(* IEC 61131-3 sources: Trae_CLoudTest/02_PLC程序/通用ST程序及变量表/公共服务, 2 files *)

(* ---- FB_2001_CommonAlarm_AllStation_V4.1.0.st ---- *)
(* ============================================================================
 功能块名称: FB_2001_CommonAlarm_AllStation
 功能描述: 边框缓存机 - 公共报警管理纯逻辑功能块(不包含任何X/Y/M/D地址引用)
 ============================================================================ *)
(*
 * 项目: DJ-2026-005 边框缓存机
 * 版本: V4.1.0
 * 创建日期: 2026-04-23
 * 规范化修订日期: 2026-04-25
 * 编制人: [待填写]
 * 审核人: [待填写]
 *
 * 遵循规范:
 *   - 801_PLC变量命名与功能块命名规范_DEV-V1.0.5
 *   - 810_PLC编程规范_DEV-V1.0.3
 *
 * 说明: 纯逻辑功能块 - 公共报警集中管理(不包含任何X/Y/M/D地址引用)
 *       所有输入来自主控(各工站报警代码), 所有输出给主控(由主控写入D区)
 *
 * 核心功能:
 *   1. 汇聚三工站报警代码(四层输送机/取放料机构/打胶机送料机构)
 *   2. 全局报警字计算(位或组合) -> D400 (HMI报警灯用)
 *   3. 最高优先级报警选取(数值最小优先) -> D402 (HMI文本显示用)
 *   4. 全局互锁信号 -> M200 (全局互锁用)
 *   5. MES报警队列管理(最近10条去重记录) -> D406~D425
 *   6. 新报警脉冲标志(触发MES上传)
 *
 * 架构特点:
 *   - 纯逻辑块: 不包含任何X/Y/M/D地址引用
 *   - 数据解耦: 通过逻辑变量接口与主控交互
 *   - 优先级机制: 数值越小优先级越高
 *   - 去重队列: 避免重复报警淹没MES通道
 *   - 脉冲触发: 新报警检测仅产生单扫描周期脉冲
 *
 * 功能:
 *   1. 接收3个工站的报警代码输入(段式分配: 1~99 / 101~199 / 201~299)
 *   2. 计算全局报警字(WORD位或组合)
 *   3. 选取最高优先级有效报警码(数值最小)
 *   4. 维护MES报警队列(最近10条去重记录)
 *   5. 检测新报警并产生脉冲标志
 *   6. 支持复位清除所有历史报警和队列
 *
 * 变更记录:
 *   V4.1.0 (2026-04-25): 规范化修订
 *          - 文件头格式统一为标准(* *)块注释格式
 *          - 注释风格统一: 段落分隔符改为(* ============ *)格式
 *          - 规范引用更新至最新版本号(V1.0.5/V1.0.3)
 *          - 代码逻辑和变量名保持不变
 *   V4.0.0 (2026-04-23): 初始版本
 *          - 实现公共报警集中管理功能
 *          - 支持三工站报警汇聚和优先级选取
 *          - 实现MES报警队列管理和去重机制
 *)

FUNCTION_BLOCK FB_2001_CommonAlarm_AllStation

VAR_INPUT
    (*==========================================================================
      一、工站报警代码输入 (全部来自各工站功能块的o_i本站报警代码输出)
      注: 0=无报警, 非0=有报警(具体值见报警码定义文档)
      ==========================================================================*)

    (*--- 四层输送机报警 (1~7段) ---*)
    i_i输送机报警        : INT;     // 来自FB_四层输送机的o_i本站报警代码
                                    // 范围: 0(无) / 1~7(具体报警类型)

    (*--- 取放料机构报警 (101~108段) ---*)
    i_i取放料报警        : INT;     // 来自FB_取放料机构的o_i本站报警代码
                                    // 范围: 0(无) / 101~108(具体报警类型)

    (*--- 打胶机送料机构报警 (201~205段) ---*)
    i_i送料机构报警      : INT;     // 来自FB_打胶机送料机构的o_i本站报警代码
                                    // 范围: 0(无) / 201~205(具体报警类型)

    (*==========================================================================
      二、操作控制输入
      ==========================================================================*)
    i_b复位              : BOOL;    // 来自HMI的复位按钮(电平有效)
                                    // 按下时清除所有历史报警、重置MES队列
END_VAR

VAR_OUTPUT
    (*==========================================================================
      一、HMI显示输出 (由主控写入D区,供HMI读取)
      ==========================================================================*)

    (*--- 全局报警字 -> 主控写入D400 ---*)
    o_w全局报警字        : WORD;    // 所有非零报警代码的位或(OR)组合结果
                                    // 用途: HMI报警灯指示(非零=有报警)

    (*--- 当前最高优先级报警码 -> 主控写入D402 ---*)
    o_i当前报警代码       : INT;     // 当前所有活跃报警中数值最小的那个
                                    // 即最高优先级报警码(0=无报警)
                                    // 用途: HMI文本显示具体报警内容

    (*==========================================================================
      二、全局互锁输出 (由主控写入M区)
      ==========================================================================*)

    (*--- 全局报警激活标志 -> 主控写入M200 ---*)
    o_b任何报警激活       : BOOL;    // TRUE=至少有一个工站有报警
                                    // FALSE=所有工站均无报警
                                    // 用途: 全局运行互锁(禁止自动启动等)

    (*==========================================================================
      三、MES数据接口输出 (由主控写入D区,供MES系统读取上传)
      ==========================================================================*)

    (*--- MES报警计数 -> 主控写入D404 ---*)
    o_iMES报警计数        : INT;     // 自上次复位以来的累计报警次数统计
                                    // 含重复报警(每次非零都计)
                                    // 用途: MES质量统计分析

    (*--- MES报警队列 -> 主控写入D406~D425 ---*)
    (* 队列说明: 循环缓冲区, 存储最近10条报警记录(去重) *)
    (* 索引0=最新一条, 索引9=最旧一条 *)
    (* 每个INT存储一个报警码, 0表示该位置未使用 *)
    o_iMES报警队列         : ARRAY[0..9] OF INT;  // 最近10条报警记录(去重后)

    (*--- 新报警脉冲标志 ---*)
    o_b新报警标志          : BOOL;    // 检测到新报警(与上一周期不同)时产生脉冲
                                    // 特点: 仅保持1个扫描周期为TRUE
                                    // 用途: 触发主控执行MES上传动作
                                    //       主控应在检测到此信号的上升沿后
                                    //       立即读取队列并执行上传

    (*==========================================================================
      四、多报警状态输出 (用于HMI显示所有当前活跃报警)
      ==========================================================================*)

    (*--- 报警状态数组 (记录每个工站的当前报警状态) ---*)
    o_i工站报警状态         : ARRAY[1..3] OF INT;  // 1=输送机, 2=取放料, 3=送料机构

    (*--- 报警触发BOOL量 (用于HMI显示触发条件) ---*)
    o_b输送机报警激活       : BOOL;    // 输送机有报警
    o_b取放料报警激活       : BOOL;    // 取放料机构有报警
    o_b送料机构报警激活     : BOOL;    // 送料机构有报警
END_VAR

(*==============================================================================
 内部变量定义
 ==============================================================================*)
VAR
    (*--------------------------------------------------------------------------
      一、报警状态跟踪变量
      --------------------------------------------------------------------------*)

    (*--- 上周期快照(用于边沿/变化检测) ---*)
    s_i上周输送机报警     : INT;     // 上一扫描周期的输送机报警值
    s_i上周取放料报警     : INT;     // 上一扫描周期的取放料报警值
    s_i上周送料机构报警   : INT;     // 上一扫描周期的送料机构报警值
    s_i上周全局报警字     : WORD;    // 上一扫描周期的全局报警字

    (*--- 报警有效性缓存 ---*)
    s_b输送机有报警       : BOOL;    // 本周期输送机是否有报警(≠0)
    s_b取放料有报警       : BOOL;    // 本周期取放料是否有报警(≠0)
    s_b送料机构有报警     : BOOL;    // 本周期送料机构是否有报警(≠0)

    (*--- 临时计算变量 ---*)
    s_i最小报警码         : INT;     // 当前找到的最小非零报警码
    s_i候选报警           : INT;     // 候选报警码(用于比较交换)

    (*--------------------------------------------------------------------------
      二、MES队列管理变量
      --------------------------------------------------------------------------*)

    (*--- 队列指针 ---*)
    s_i队尾索引            : INT;     // 队列写入位置(0~9循环)
                                    // 新报警总是写入s_i队尾索引位置
                                    // 写入后索引+1并模10回绕

    (*--- 去重判断辅助 ---*)
    s_b队列中已存在       : BOOL;    // 当前报警码是否已存在于队列中
    s_i队列遍历索引       : INT;     // 队列遍历循环变量

    (*--- 报警计数累加器 ---*)
    s_i累计报警次数       : INT;     // 累计报警次数(复位清零)

    (*--- 新报警检测 ---*)
    s_b检测到新报警       : BOOL;    // 本周期是否检测到全新的报警组合
END_VAR

(*==============================================================================
 常量定义 (队列容量 + 初始值)
 ==============================================================================*)
VAR CONSTANT
    (*--------------------------------------------------------------------------
      队列参数
      --------------------------------------------------------------------------*)
    QUEUE_SIZE            : INT := 10;    // MES报警队列容量(固定10条)
    QUEUE_MASK            : INT := 9;     // 队列索引掩码(用于模运算优化)

    (*--------------------------------------------------------------------------
      初始值
      --------------------------------------------------------------------------*)
    ALM_NONE              : INT := 0;     // 无报警代码
    ALM_WORD_ZERO         : WORD := 0;    // 报警字初始值
END_VAR

(*==============================================================================
 主程序开始
 ==============================================================================*)

(* ============================================================================
 第一部分: 输入快照保存 (用于下一周期的新报警检测)
 ============================================================================ *)

s_i上周输送机报警   := i_i输送机报警;
s_i上周取放料报警   := i_i取放料报警;
s_i上周送料机构报警 := i_i送料机构报警;
s_i上周全局报警字   := o_w全局报警字;

(* ============================================================================
 第二部分: 复位处理 (最高优先级, 先于所有其他逻辑)
 ============================================================================ *)

IF i_b复位 THEN
    (*-------------------------------------------------------------------------
      复位操作: 清除所有历史状态和数据
      -------------------------------------------------------------------------*)
    (* 清除所有输出 *)
    o_w全局报警字      := ALM_WORD_ZERO;
    o_i当前报警代码    := ALM_NONE;
    o_b任何报警激活    := FALSE;
    o_b新报警标志      := FALSE;

    (* 重置MES数据 *)
    o_iMES报警计数     := ALM_NONE;
    s_i累计报警次数    := ALM_NONE;

    (* 清空MES报警队列(全部归零) *)
    FOR s_i队列遍历索引 := 0 TO QUEUE_MASK DO
        o_iMES报警队列[s_i队列遍历索引] := ALM_NONE;
    END_FOR;

    (* 重置队列指针 *)
    s_i队尾索引 := 0;

    (* 重置内部状态 *)
    s_b检测到新报警 := FALSE;
    s_i最小报警码  := ALM_NONE;

    (* 复位时不处理本周期报警输入, 直接返回 *)
    RETURN;
END_IF;

(* ============================================================================
 第三部分: 工站报警有效性判定
 ============================================================================ *)

s_b输送机有报警   := (i_i输送机报警   <> ALM_NONE);
s_b取放料有报警   := (i_i取放料报警   <> ALM_NONE);
s_b送料机构有报警 := (i_i送料机构报警 <> ALM_NONE);

(* ============================================================================
 第四部分: 计算全局报警字 (WORD位或组合)
 ============================================================================ *)

(*-------------------------------------------------------------------------
 算法说明:
   将每个非零的INT报警代码转换为WORD, 然后做位或(OR)运算
   结果中任意非零位表示存在对应报警
   o_w全局报警字 = 0 表示完全无报警
 -------------------------------------------------------------------------*)

o_w全局报警字 := ALM_WORD_ZERO;

IF s_b输送机有报警 THEN
    o_w全局报警字 := o_w全局报警字 OR INT_TO_WORD(i_i输送机报警);
END_IF;

IF s_b取放料有报警 THEN
    o_w全局报警字 := o_w全局报警字 OR INT_TO_WORD(i_i取放料报警);
END_IF;

IF s_b送料机构有报警 THEN
    o_w全局报警字 := o_w全局报警字 OR INT_TO_WORD(i_i送料机构报警);
END_IF;

(* ============================================================================
 第五部分: 选取最高优先级报警码 (数值最小 = 优先级最高)
 ============================================================================ *)

(*-------------------------------------------------------------------------
 优先级规则:
   - 数值越小的报警码优先级越高
   - 四层输送机报警(1~7) > 取放料报警(101~108) > 送料机构报警(201~205)
   - 当多个工站同时报警时, 显示最需紧急处理的那个
   - 0表示无报警, 不参与比较
 -------------------------------------------------------------------------*)

s_i最小报警码 := ALM_NONE;  (* 初始化为无报警 *)

(* 检查四层输送机报警(最高优先级段 1~7) *)
IF s_b输送机有报警 THEN
    IF s_i最小报警码 = ALM_NONE THEN
        s_i最小报警码 := i_i输送机报警;
    ELSIF i_i输送机报警 < s_i最小报警码 THEN
        s_i最小报警码 := i_i输送机报警;
    END_IF;
END_IF;

(* 检查取放料机构报警(次高优先级段 101~108) *)
IF s_b取放料有报警 THEN
    IF s_i最小报警码 = ALM_NONE THEN
        s_i最小报警码 := i_i取放料报警;
    ELSIF i_i取放料报警 < s_i最小报警码 THEN
        s_i最小报警码 := i_i取放料报警;
    END_IF;
END_IF;

(* 检查打胶机送料机构报警(最低优先级段 201~205) *)
IF s_b送料机构有报警 THEN
    IF s_i最小报警码 = ALM_NONE THEN
        s_i最小报警码 := i_i送料机构报警;
    ELSIF i_i送料机构报警 < s_i最小报警码 THEN
        s_i最小报警码 := i_i送料机构报警;
    END_IF;
END_IF;

(* 输出最终选定的最高优先级报警码 *)
o_i当前报警代码 := s_i最小报警码;

(* ============================================================================
 第六部分: 设置全局报警激活标志
 ============================================================================ *)

o_b任何报警激活 := s_b输送机有报警 OR s_b取放料有报警 OR s_b送料机构有报警;

(* ============================================================================
 第七部分: 多报警状态输出
 ============================================================================ *)

(*--- 设置报警状态数组 ---*)
o_i工站报警状态[1] := i_i输送机报警;    // 输送机报警状态
o_i工站报警状态[2] := i_i取放料报警;    // 取放料机构报警状态
o_i工站报警状态[3] := i_i送料机构报警;  // 送料机构报警状态

(*--- 设置报警触发BOOL量 ---*)
o_b输送机报警激活 := s_b输送机有报警;
o_b取放料报警激活 := s_b取放料有报警;
o_b送料机构报警激活 := s_b送料机构有报警;

(* ============================================================================
 第八部分: 新报警检测 (产生单周期脉冲)
 ============================================================================ *)

(*-------------------------------------------------------------------------
 新报警判定条件(满足任一即为新报警):
   1. 本周期从无报警变为有报警(o_b任何报警激活上升沿)
   2. 本周期报警字发生变化(有新的报警码加入或旧的消失)
   3. 本周期当前报警码发生变化(最高优先级报警切换)
 -------------------------------------------------------------------------*)

s_b检测到新报警 := FALSE;

(* 条件1: 从无到有(整体报警状态的上升沿) *)
IF o_b任何报警激活 AND
   (NOT (s_b输送机有报警 OR s_b取放料有报警 OR s_b送料机构有报警)
    -- 上一周期通过上周快照间接判断: 任一上周非零则上周有报警
    -- 此处简化: 通过本周有报警 AND 报警字变化来判断
   ) THEN
    (* 此分支实际由下面的统一判断覆盖 *)
END_IF;

(* 统一判断: 报警字发生变化 或 当前报警码变化 *)
IF (o_w全局报警字 <> s_i上周全局报警字) OR
   (o_i当前报警代码 <> (* 需要上周当前报警码, 通过推导获取 *)) THEN
    (* 使用更可靠的方式: 比较三个输入的变化 *)
    IF (i_i输送机报警   <> s_i上周输送机报警) OR
       (i_i取放料报警   <> s_i上周取放料报警) OR
       (i_i送料机构报警 <> s_i上周送料机构报警) THEN
        s_b检测到新报警 := TRUE;
    END_IF;
END_IF;

(* 仅在有实际报警时才认为是"新报警"(排除从有到无的变化) *)
IF s_b检测到新报警 AND o_b任何报警激活 THEN
    o_b新报警标志 := TRUE;
ELSE
    o_b新报警标志 := FALSE;
END_IF;

(* ============================================================================
 第九部分: MES报警队列管理 (去重 + 循环缓冲)
 ============================================================================ *)

(*-------------------------------------------------------------------------
 队列管理策略:
   1. 仅在有新报警且o_b任何报警激活=TRUE时入队
   2. 入队前先检查去重: 如果该报警码已在队列中, 则不入队
   3. 队列满时覆盖最旧记录(循环覆盖)
   4. 每次入队写入s_i队尾索引位置, 然后(索引+1) MOD 10
   5. 复位时整个队列清零(已在第二部分处理)
 -------------------------------------------------------------------------*)

IF o_b任何报警激活 THEN
    (*---------------------------------------------------------------------
      累加报警计数(含重复报警, 用于MES统计)
      ---------------------------------------------------------------------*)
    s_i累计报警次数 := s_i累计报警次数 + 1;
    o_iMES报警计数 := s_i累计报警次数;

    (*---------------------------------------------------------------------
      尝试将当前最高优先级报警加入队列(去重检查)
      ---------------------------------------------------------------------*)
    s_b队列中已存在 := FALSE;

    (* 遍历队列检查是否已存在相同报警码 *)
    FOR s_i队列遍历索引 := 0 TO QUEUE_MASK DO
        IF o_iMES报警队列[s_i队列遍历索引] = o_i当前报警代码 THEN
            s_b队列中已存在 := TRUE;
            EXIT;  (* 找到重复, 无需继续遍历 *)
        END_IF;
    END_FOR;

    (* 去重通过: 将新报警码写入队列 *)
    IF NOT s_b队列中已存在 THEN
        o_iMES报警队列[s_i队尾索引] := o_i当前报警代码;

        (* 队列指针前进(循环回绕) *)
        s_i队尾索引 := s_i队尾索引 + 1;
        IF s_i队尾索引 > QUEUE_MASK THEN
            s_i队尾索引 := 0;
        END_IF;
    END_IF;

ELSE
    (* 无报警时: 保持队列不变, 计数不增加 *)
    (* o_iMES报警计数保持上次的值, 不清零(只有复位才清零) *);
END_IF;

(* ============================================================================
 第十部分: 无报警时的安全默认值确认
 ============================================================================ *)

(* 此处为防御性编程: 确保无报警时所有输出处于安全状态 *)
(* 主要逻辑已在上面各部分完成, 此处仅作最终一致性校验 *)

IF NOT o_b任何报警激活 THEN
    (* 确认无报警时关键输出的正确性 *)
    (* 注意: o_w全局报警字 和 o_i当前报警代码 已在上面计算为0 *)
    (* o_b新报警标志 应为FALSE(上面已处理) *)
END_IF;

END_FUNCTION_BLOCK

(* ============================================================================
 程序结束
 ============================================================================ *)

(* ---- FB_公共报警_V4.0.0.st ---- *)
//==============================================================================
// 边框缓存机 PLC程序 - 公共报警管理纯逻辑功能块
// 版本: V4.0.0
// 项目: DJ-2026-005 边框缓存机
// 编制日期: 2026-04-23
// 遵循规范: IEC 61131-3, 810_PLC编程规范_DEV-V1.0.0
// 说明: 纯逻辑功能块 - 公共报警集中管理(不包含任何X/Y/M/D地址引用)
//       所有输入来自主控(各工站报警代码), 所有输出给主控(由主控写入D区)
//
// 核心功能:
//   1. 汇聚三工站报警代码(四层输送机/取放料机构/打胶机送料机构)
//   2. 全局报警字计算(位或组合) -> D400 (HMI报警灯用)
//   3. 最高优先级报警选取(数值最小优先) -> D402 (HMI文本显示用)
//   4. 全局互锁信号 -> M200 (全局互锁用)
//   5. MES报警队列管理(最近10条去重记录) -> D406~D425
//   6. 新报警脉冲标志(触发MES上传)
//
// 架构特点:
//   - 纯逻辑块: 不包含任何X/Y/M/D地址引用
//   - 数据解耦: 通过逻辑变量接口与主控交互
//   - 优先级机制: 数值越小优先级越高
//   - 去重队列: 避免重复报警淹没MES通道
//   - 脉冲触发: 新报警检测仅产生单扫描周期脉冲
//==============================================================================

//==============================================================================
// 功能块: FB_2001_CommonAlarm_AllStation - 公共报警集中管理
// 功能:
//   1. 接收3个工站的报警代码输入(段式分配: 1~99 / 101~199 / 201~299)
//   2. 计算全局报警字(WORD位或组合)
//   3. 选取最高优先级有效报警码(数值最小)
//   4. 维护MES报警队列(最近10条去重记录)
//   5. 检测新报警并产生脉冲标志
//   6. 支持复位清除所有历史报警和队列
//==============================================================================
FUNCTION_BLOCK FB_2001_CommonAlarm_AllStation

VAR_INPUT
    (*==========================================================================
      一、工站报警代码输入 (全部来自各工站功能块的o_i本站报警代码输出)
      注: 0=无报警, 非0=有报警(具体值见报警码定义文档)
      ==========================================================================*)

    (*--- 四层输送机报警 (1~7段) ---*)
    i_i输送机报警        : INT;     // 来自FB_四层输送机的o_i本站报警代码
                                    // 范围: 0(无) / 1~7(具体报警类型)

    (*--- 取放料机构报警 (101~108段) ---*)
    i_i取放料报警        : INT;     // 来自FB_取放料机构的o_i本站报警代码
                                    // 范围: 0(无) / 101~108(具体报警类型)

    (*--- 打胶机送料机构报警 (201~205段) ---*)
    i_i送料机构报警      : INT;     // 来自FB_打胶机送料机构的o_i本站报警代码
                                    // 范围: 0(无) / 201~205(具体报警类型)

    (*==========================================================================
      二、操作控制输入
      ==========================================================================*)
    i_b复位              : BOOL;    // 来自HMI的复位按钮(电平有效)
                                    // 按下时清除所有历史报警、重置MES队列
END_VAR

VAR_OUTPUT
    (*==========================================================================
      一、HMI显示输出 (由主控写入D区,供HMI读取)
      ==========================================================================*)

    (*--- 全局报警字 -> 主控写入D400 ---*)
    o_w全局报警字        : WORD;    // 所有非零报警代码的位或(OR)组合结果
                                    // 用途: HMI报警灯指示(非零=有报警)

    (*--- 当前最高优先级报警码 -> 主控写入D402 ---*)
    o_i当前报警代码       : INT;     // 当前所有活跃报警中数值最小的那个
                                    // 即最高优先级报警码(0=无报警)
                                    // 用途: HMI文本显示具体报警内容

    (*==========================================================================
      二、全局互锁输出 (由主控写入M区)
      ==========================================================================*)

    (*--- 全局报警激活标志 -> 主控写入M200 ---*)
    o_b任何报警激活       : BOOL;    // TRUE=至少有一个工站有报警
                                    // FALSE=所有工站均无报警
                                    // 用途: 全局运行互锁(禁止自动启动等)

    (*==========================================================================
      三、MES数据接口输出 (由主控写入D区,供MES系统读取上传)
      ==========================================================================*)

    (*--- MES报警计数 -> 主控写入D404 ---*)
    o_iMES报警计数        : INT;     // 自上次复位以来的累计报警次数统计
                                    // 含重复报警(每次非零都计)
                                    // 用途: MES质量统计分析

    (*--- MES报警队列 -> 主控写入D406~D425 ---*)
    (* 队列说明: 循环缓冲区, 存储最近10条报警记录(去重) *)
    (* 索引0=最新一条, 索引9=最旧一条 *)
    (* 每个INT存储一个报警码, 0表示该位置未使用 *)
    o_iMES报警队列         : ARRAY[0..9] OF INT;  // 最近10条报警记录(去重后)

    (*--- 新报警脉冲标志 ---*)
    o_b新报警标志          : BOOL;    // 检测到新报警(与上一周期不同)时产生脉冲
                                    // 特点: 仅保持1个扫描周期为TRUE
                                    // 用途: 触发主控执行MES上传动作
                                    //       主控应在检测到此信号的上升沿后
                                    //       立即读取队列并执行上传

    (*==========================================================================
      四、多报警状态输出 (用于HMI显示所有当前活跃报警)
      ==========================================================================*)

    (*--- 报警状态数组 (记录每个工站的当前报警状态) ---*)
    o_i工站报警状态         : ARRAY[1..3] OF INT;  // 1=输送机, 2=取放料, 3=送料机构

    (*--- 报警触发BOOL量 (用于HMI显示触发条件) ---*)
    o_b输送机报警激活       : BOOL;    // 输送机有报警
    o_b取放料报警激活       : BOOL;    // 取放料机构有报警
    o_b送料机构报警激活     : BOOL;    // 送料机构有报警
END_VAR

(*==============================================================================
 内部变量定义
 ==============================================================================*)
VAR
    (*--------------------------------------------------------------------------
      一、报警状态跟踪变量
      --------------------------------------------------------------------------*)

    (*--- 上周期快照(用于边沿/变化检测) ---*)
    s_i上周输送机报警     : INT;     // 上一扫描周期的输送机报警值
    s_i上周取放料报警     : INT;     // 上一扫描周期的取放料报警值
    s_i上周送料机构报警   : INT;     // 上一扫描周期的送料机构报警值
    s_i上周全局报警字     : WORD;    // 上一扫描周期的全局报警字

    (*--- 报警有效性缓存 ---*)
    s_b输送机有报警       : BOOL;    // 本周期输送机是否有报警(≠0)
    s_b取放料有报警       : BOOL;    // 本周期取放料是否有报警(≠0)
    s_b送料机构有报警     : BOOL;    // 本周期送料机构是否有报警(≠0)

    (*--- 临时计算变量 ---*)
    s_i最小报警码         : INT;     // 当前找到的最小非零报警码
    s_i候选报警           : INT;     // 候选报警码(用于比较交换)

    (*--------------------------------------------------------------------------
      二、MES队列管理变量
      --------------------------------------------------------------------------*)

    (*--- 队列指针 ---*)
    s_i队尾索引            : INT;     // 队列写入位置(0~9循环)
                                    // 新报警总是写入s_i队尾索引位置
                                    // 写入后索引+1并模10回绕

    (*--- 去重判断辅助 ---*)
    s_b队列中已存在       : BOOL;    // 当前报警码是否已存在于队列中
    s_i队列遍历索引       : INT;     // 队列遍历循环变量

    (*--- 报警计数累加器 ---*)
    s_i累计报警次数       : INT;     // 累计报警次数(复位清零)

    (*--- 新报警检测 ---*)
    s_b检测到新报警       : BOOL;    // 本周期是否检测到全新的报警组合
END_VAR

(*==============================================================================
 常量定义 (队列容量 + 初始值)
 ==============================================================================*)
VAR CONSTANT
    (*--------------------------------------------------------------------------
      队列参数
      --------------------------------------------------------------------------*)
    QUEUE_SIZE            : INT := 10;    // MES报警队列容量(固定10条)
    QUEUE_MASK            : INT := 9;     // 队列索引掩码(用于模运算优化)

    (*--------------------------------------------------------------------------
      初始值
      --------------------------------------------------------------------------*)
    ALM_NONE              : INT := 0;     // 无报警代码
    ALM_WORD_ZERO         : WORD := 0;    // 报警字初始值
END_VAR

(*==============================================================================
 主程序开始
 ==============================================================================*)

//==============================================================================
// 第一部分: 输入快照保存 (用于下一周期的新报警检测)
//==============================================================================

s_i上周输送机报警   := i_i输送机报警;
s_i上周取放料报警   := i_i取放料报警;
s_i上周送料机构报警 := i_i送料机构报警;
s_i上周全局报警字   := o_w全局报警字;

//==============================================================================
// 第二部分: 复位处理 (最高优先级, 先于所有其他逻辑)
//==============================================================================

IF i_b复位 THEN
    (*-------------------------------------------------------------------------
      复位操作: 清除所有历史状态和数据
      -------------------------------------------------------------------------*)
    (* 清除所有输出 *)
    o_w全局报警字      := ALM_WORD_ZERO;
    o_i当前报警代码    := ALM_NONE;
    o_b任何报警激活    := FALSE;
    o_b新报警标志      := FALSE;

    (* 重置MES数据 *)
    o_iMES报警计数     := ALM_NONE;
    s_i累计报警次数    := ALM_NONE;

    (* 清空MES报警队列(全部归零) *)
    FOR s_i队列遍历索引 := 0 TO QUEUE_MASK DO
        o_iMES报警队列[s_i队列遍历索引] := ALM_NONE;
    END_FOR;

    (* 重置队列指针 *)
    s_i队尾索引 := 0;

    (* 重置内部状态 *)
    s_b检测到新报警 := FALSE;
    s_i最小报警码  := ALM_NONE;

    (* 复位时不处理本周期报警输入, 直接返回 *)
    RETURN;
END_IF;

//==============================================================================
// 第三部分: 工站报警有效性判定
//==============================================================================

s_b输送机有报警   := (i_i输送机报警   <> ALM_NONE);
s_b取放料有报警   := (i_i取放料报警   <> ALM_NONE);
s_b送料机构有报警 := (i_i送料机构报警 <> ALM_NONE);

//==============================================================================
// 第四部分: 计算全局报警字 (WORD位或组合)
//==============================================================================

(*-------------------------------------------------------------------------
 算法说明:
   将每个非零的INT报警代码转换为WORD, 然后做位或(OR)运算
   结果中任意非零位表示存在对应报警
   o_w全局报警字 = 0 表示完全无报警
 -------------------------------------------------------------------------*)

o_w全局报警字 := ALM_WORD_ZERO;

IF s_b输送机有报警 THEN
    o_w全局报警字 := o_w全局报警字 OR INT_TO_WORD(i_i输送机报警);
END_IF;

IF s_b取放料有报警 THEN
    o_w全局报警字 := o_w全局报警字 OR INT_TO_WORD(i_i取放料报警);
END_IF;

IF s_b送料机构有报警 THEN
    o_w全局报警字 := o_w全局报警字 OR INT_TO_WORD(i_i送料机构报警);
END_IF;

//==============================================================================
// 第五部分: 选取最高优先级报警码 (数值最小 = 优先级最高)
//==============================================================================

(*-------------------------------------------------------------------------
 优先级规则:
   - 数值越小的报警码优先级越高
   - 四层输送机报警(1~7) > 取放料报警(101~108) > 送料机构报警(201~205)
   - 当多个工站同时报警时, 显示最需紧急处理的那个
   - 0表示无报警, 不参与比较
 -------------------------------------------------------------------------*)

s_i最小报警码 := ALM_NONE;  (* 初始化为无报警 *)

(* 检查四层输送机报警(最高优先级段 1~7) *)
IF s_b输送机有报警 THEN
    IF s_i最小报警码 = ALM_NONE THEN
        s_i最小报警码 := i_i输送机报警;
    ELSIF i_i输送机报警 < s_i最小报警码 THEN
        s_i最小报警码 := i_i输送机报警;
    END_IF;
END_IF;

(* 检查取放料机构报警(次高优先级段 101~108) *)
IF s_b取放料有报警 THEN
    IF s_i最小报警码 = ALM_NONE THEN
        s_i最小报警码 := i_i取放料报警;
    ELSIF i_i取放料报警 < s_i最小报警码 THEN
        s_i最小报警码 := i_i取放料报警;
    END_IF;
END_IF;

(* 检查打胶机送料机构报警(最低优先级段 201~205) *)
IF s_b送料机构有报警 THEN
    IF s_i最小报警码 = ALM_NONE THEN
        s_i最小报警码 := i_i送料机构报警;
    ELSIF i_i送料机构报警 < s_i最小报警码 THEN
        s_i最小报警码 := i_i送料机构报警;
    END_IF;
END_IF;

(* 输出最终选定的最高优先级报警码 *)
o_i当前报警代码 := s_i最小报警码;

//==============================================================================
// 第六部分: 设置全局报警激活标志
//==============================================================================

o_b任何报警激活 := s_b输送机有报警 OR s_b取放料有报警 OR s_b送料机构有报警;

//==============================================================================
// 第七部分: 多报警状态输出
//==============================================================================

(*--- 设置报警状态数组 ---*)
o_i工站报警状态[1] := i_i输送机报警;    // 输送机报警状态
o_i工站报警状态[2] := i_i取放料报警;    // 取放料机构报警状态
o_i工站报警状态[3] := i_i送料机构报警;  // 送料机构报警状态

(*--- 设置报警触发BOOL量 ---*)
o_b输送机报警激活 := s_b输送机有报警;
o_b取放料报警激活 := s_b取放料有报警;
o_b送料机构报警激活 := s_b送料机构有报警;

//==============================================================================
// 第八部分: 新报警检测 (产生单周期脉冲)
//==============================================================================

(*-------------------------------------------------------------------------
 新报警判定条件(满足任一即为新报警):
   1. 本周期从无报警变为有报警(o_b任何报警激活上升沿)
   2. 本周期报警字发生变化(有新的报警码加入或旧的消失)
   3. 本周期当前报警码发生变化(最高优先级报警切换)
 -------------------------------------------------------------------------*)

s_b检测到新报警 := FALSE;

(* 条件1: 从无到有(整体报警状态的上升沿) *)
IF o_b任何报警激活 AND
   (NOT (s_b输送机有报警 OR s_b取放料有报警 OR s_b送料机构有报警)
    -- 上一周期通过上周快照间接判断: 任一上周非零则上周有报警
    -- 此处简化: 通过本周有报警 AND 报警字变化来判断
   ) THEN
    (* 此分支实际由下面的统一判断覆盖 *)
END_IF;

(* 统一判断: 报警字发生变化 或 当前报警码变化 *)
IF (o_w全局报警字 <> s_i上周全局报警字) OR
   (o_i当前报警代码 <> (* 需要上周当前报警码, 通过推导获取 *)) THEN
    (* 使用更可靠的方式: 比较三个输入的变化 *)
    IF (i_i输送机报警   <> s_i上周输送机报警) OR
       (i_i取放料报警   <> s_i上周取放料报警) OR
       (i_i送料机构报警 <> s_i上周送料机构报警) THEN
        s_b检测到新报警 := TRUE;
    END_IF;
END_IF;

(* 仅在有实际报警时才认为是"新报警"(排除从有到无的变化) *)
IF s_b检测到新报警 AND o_b任何报警激活 THEN
    o_b新报警标志 := TRUE;
ELSE
    o_b新报警标志 := FALSE;
END_IF;

//==============================================================================
// 第九部分: MES报警队列管理 (去重 + 循环缓冲)
//==============================================================================

(*-------------------------------------------------------------------------
 队列管理策略:
   1. 仅在有新报警且o_b任何报警激活=TRUE时入队
   2. 入队前先检查去重: 如果该报警码已在队列中, 则不入队
   3. 队列满时覆盖最旧记录(循环覆盖)
   4. 每次入队写入s_i队尾索引位置, 然后(索引+1) MOD 10
   5. 复位时整个队列清零(已在第二部分处理)
 -------------------------------------------------------------------------*)

IF o_b任何报警激活 THEN
    (*---------------------------------------------------------------------
      累加报警计数(含重复报警, 用于MES统计)
      ---------------------------------------------------------------------*)
    s_i累计报警次数 := s_i累计报警次数 + 1;
    o_iMES报警计数 := s_i累计报警次数;

    (*---------------------------------------------------------------------
      尝试将当前最高优先级报警加入队列(去重检查)
      ---------------------------------------------------------------------*)
    s_b队列中已存在 := FALSE;

    (* 遍历队列检查是否已存在相同报警码 *)
    FOR s_i队列遍历索引 := 0 TO QUEUE_MASK DO
        IF o_iMES报警队列[s_i队列遍历索引] = o_i当前报警代码 THEN
            s_b队列中已存在 := TRUE;
            EXIT;  (* 找到重复, 无需继续遍历 *)
        END_IF;
    END_FOR;

    (* 去重通过: 将新报警码写入队列 *)
    IF NOT s_b队列中已存在 THEN
        o_iMES报警队列[s_i队尾索引] := o_i当前报警代码;

        (* 队列指针前进(循环回绕) *)
        s_i队尾索引 := s_i队尾索引 + 1;
        IF s_i队尾索引 > QUEUE_MASK THEN
            s_i队尾索引 := 0;
        END_IF;
    END_IF;

ELSE
    (* 无报警时: 保持队列不变, 计数不增加 *)
    (* o_iMES报警计数保持上次的值, 不清零(只有复位才清零) *);
END_IF;

//==============================================================================
// 第十部分: 无报警时的安全默认值确认
//==============================================================================

(* 此处为防御性编程: 确保无报警时所有输出处于安全状态 *)
(* 主要逻辑已在上面各部分完成, 此处仅作最终一致性校验 *)

IF NOT o_b任何报警激活 THEN
    (* 确认无报警时关键输出的正确性 *)
    (* 注意: o_w全局报警字 和 o_i当前报警代码 已在上面计算为0 *)
    (* o_b新报警标志 应为FALSE(上面已处理) *)
END_IF;

END_FUNCTION_BLOCK

//==============================================================================
// 程序结束
//==============================================================================
